(* IEC 61131-3 sources: eCockpitGit/test_project/src/%F%00 Library/%F%JSON/%POU%FB_JSONReader/%F%Read, 13 files *)

(* ---- %METH%compareString.st ---- *)
//Returns true if the inputted string is the same as the read string
METHOD compareString : BOOL
VAR_INPUT
	str				:POINTER TO EASCII;
END_VAR
VAR
	posBuffer		:POINTER TO EASCII := lastValueStart + 1;		//Buffer for key position
END_VAR
(*%!%__DELIMITER__%!%*)
IF ready AND_THEN lastValueType = EStructType.tString THEN
	WHILE posBuffer <= bufferADRMax DO
		CASE posBuffer^ OF
			EASCII.Null:
				compareString			:=		str^ = EASCII.Null;
				EXIT;
			EASCII.DoubleQoute:
				IF checkNoBackSlash(checkPos:=posBuffer) THEN
					compareString		:=		str^ = EASCII.Null;
					EXIT;
				END_IF
		END_CASE
		IF str^ <> posBuffer^ THEN
			IF posBuffer^ = EASCII.BackSlash THEN
				posBuffer				:=		posBuffer + 1;
				IF str^ <> posBuffer^ THEN
					EXIT;
				END_IF
			ELSE
				EXIT;
			END_IF
		END_IF
		str								:=		str + 1;
		posBuffer						:=		posBuffer + 1;
	END_WHILE
END_IF

(* ---- %METH%exportValue.st ---- *)
//This method outputs the start address and size of the current value
//True when ok
// |**Version**|**Author**| **Date** |**Changes**
// | 1         | NSN      | 04-06-18 | Creation
METHOD exportValue : BOOL
VAR_OUTPUT
	position		:POINTER TO EASCII;
	size			:DWORD;
END_VAR
VAR
	inString		:BOOL;
	posBuffer		:POINTER TO EASCII := lastValueStart;
	level			:WORD := 1;		//This value makes sure it doesn't return a key from inside another object
END_VAR
(*%!%__DELIMITER__%!%*)
IF ready AND lastValueStart <> 0 THEN
	position					:=		lastValueStart;
	WHILE posBuffer < bufferADRMax DO
		CASE posBuffer^ OF
			EASCII.Null:
				EXIT;
			EASCII.DoubleQoute:
				IF checkNoBackSlash(checkPos:=posBuffer) THEN
					inString	:=		NOT(inString);
				END_IF
			EASCII.CloseBraces,EASCII.SqBracketC:
				IF NOT(inString) THEN
					IF level > 1 THEN
						level	:=		level - 1;
					ELSE
						EXIT;
					END_IF
				END_IF
			EASCII.Comma:
				IF NOT(inString) THEN
					IF level <= 1 THEN
						EXIT;
					END_IF
				END_IF
			EASCII.OpenBraces,EASCII.SqBracketO:
				IF NOT(inString) THEN
					level		:=		level + 1;
				END_IF
		END_CASE
		posBuffer				:=		posBuffer + 1;
	END_WHILE
	size						:=		posBuffer - position;
	exportValue					:=		TRUE;
END_IF

(* ---- %METH%readBool.st ---- *)
METHOD readBool :BOOL
VAR
	valueBuff	:STRING(30);
END_VAR
(*%!%__DELIMITER__%!%*)
IF ready THEN
	CASE lastValueType OF
		EStructType.tBool:
			readBool				:=		lastValueStart^ = EASCII.Smallt;
		EStructType.number:
			readString(str:=ADR(valueBuff),lenMax:=30);
			readBool				:=		TO_BOOL(TO_REAL(valueBuff));
		EStructType.null:;
		EStructType.object,EStructType.tArray:
			readBool				:=		amountInSelection > 0;
		EStructType.tString:
			readString(str:=ADR(valueBuff),lenMax:=5);
			readBool				:=		TO_BOOL(valueBuff);
			IF NOT(readBool) THEN
				readBool			:=		valueBuff[0] <> 0;
			END_IF
	END_CASE
END_IF

(* ---- %METH%readByte.st ---- *)
METHOD readByte : BYTE
VAR
	buffer		:STRING(30);
	posBuffer	:POINTER TO EASCII := lastValueStart;		//Buffer for key position
	i			:BYTE;
END_VAR
(*%!%__DELIMITER__%!%*)
IF ready THEN
	CASE lastValueType OF
		EStructType.tBool:
			IF lastValueStart^ = EASCII.Smallt THEN
				readByte			:=		1;
			END_IF
		EStructType.number:
			WHILE posBuffer <= bufferADRMax AND i < 31 DO
				CASE posBuffer^ OF
					EASCII.Zero,EASCII.One,EASCII.Two,EASCII.Three,EASCII.Four,EASCII.Five,EASCII.Six,EASCII.Seven,EASCII.Eight,EASCII.Nine:;
				ELSE
					EXIT;
				END_CASE
				buffer[i]			:=		posBuffer^;
				posBuffer			:=		posBuffer + 1;
				i					:=		i + 1;
			END_WHILE
			buffer[i]				:=		EASCII.Null;
			readByte				:=		TO_BYTE(buffer);
		EStructType.null,EStructType.object,EStructType.tArray:;
		EStructType.tString:
			readString(str:=ADR(buffer),lenMax:=30);
			readByte				:=		TO_BYTE(buffer);
	END_CASE
END_IF

(* ---- %METH%readDint.st ---- *)
METHOD readDint : DINT
VAR
	buffer		:STRING(30);
	posBuffer	:POINTER TO EASCII := lastValueStart;		//Buffer for key position
	i			:BYTE;
END_VAR
(*%!%__DELIMITER__%!%*)
IF ready THEN
	CASE lastValueType OF
		EStructType.tBool:
			IF lastValueStart^ = EASCII.Smallt THEN
				readDint			:=		1;
			END_IF
		EStructType.number:
			WHILE posBuffer <= bufferADRMax AND i < 31 DO
				CASE posBuffer^ OF
					EASCII.Zero,EASCII.One,EASCII.Two,EASCII.Three,EASCII.Four,EASCII.Five,EASCII.Six,EASCII.Seven,EASCII.Eight,EASCII.Nine,EASCII.Minus:;
				ELSE
					EXIT;
				END_CASE
				buffer[i]			:=		posBuffer^;
				posBuffer			:=		posBuffer + 1;
				i					:=		i + 1;
			END_WHILE
			buffer[i]				:=		EASCII.Null;
			readDint				:=		TO_DINT(buffer);
		EStructType.null,EStructType.object,EStructType.tArray:;
		EStructType.tString:
			readString(str:=ADR(buffer),lenMax:=30);
			readDint				:=		TO_DINT(buffer);
	END_CASE
END_IF

(* ---- %METH%readDword.st ---- *)
METHOD readDword : DWORD
VAR
	buffer		:STRING(30);
	posBuffer	:POINTER TO EASCII := lastValueStart;		//Buffer for key position
	i			:BYTE;
END_VAR
(*%!%__DELIMITER__%!%*)
IF ready THEN
	CASE lastValueType OF
		EStructType.tBool:
			IF lastValueStart^ = EASCII.Smallt THEN
				readDword			:=		1;
			END_IF
		EStructType.number:
			WHILE posBuffer <= bufferADRMax AND i < 31 DO
				CASE posBuffer^ OF
					EASCII.Zero,EASCII.One,EASCII.Two,EASCII.Three,EASCII.Four,EASCII.Five,EASCII.Six,EASCII.Seven,EASCII.Eight,EASCII.Nine:;
				ELSE
					EXIT;
				END_CASE
				buffer[i]			:=		posBuffer^;
				posBuffer			:=		posBuffer + 1;
				i					:=		i + 1;
			END_WHILE
			buffer[i]				:=		EASCII.Null;
			readDword				:=		TO_DWORD(buffer);
		EStructType.null,EStructType.object,EStructType.tArray:;
		EStructType.tString:
			readString(str:=ADR(buffer),lenMax:=30);
			readDword				:=		TO_DWORD(buffer);
	END_CASE
END_IF

(* ---- %METH%readInt.st ---- *)
METHOD readInt : INT
VAR
	buffer		:STRING(30);
	posBuffer	:POINTER TO EASCII := lastValueStart;		//Buffer for key position
	i			:BYTE;
END_VAR
(*%!%__DELIMITER__%!%*)
IF ready THEN
	CASE lastValueType OF
		EStructType.tBool:
			IF lastValueStart^ = EASCII.Smallt THEN
				readInt				:=		1;
			END_IF
		EStructType.number:
			WHILE posBuffer <= bufferADRMax AND i < 31 DO
				CASE posBuffer^ OF
					EASCII.Zero,EASCII.One,EASCII.Two,EASCII.Three,EASCII.Four,EASCII.Five,EASCII.Six,EASCII.Seven,EASCII.Eight,EASCII.Nine,EASCII.Minus:;
				ELSE
					EXIT;
				END_CASE
				buffer[i]			:=		posBuffer^;
				posBuffer			:=		posBuffer + 1;
				i					:=		i + 1;
			END_WHILE
			buffer[i]				:=		EASCII.Null;
			readInt					:=		TO_INT(buffer);
		EStructType.null,EStructType.object,EStructType.tArray:;
		EStructType.tString:
			readString(str:=ADR(buffer),lenMax:=30);
			readInt					:=		TO_INT(buffer);
	END_CASE
END_IF

(* ---- %METH%readLint.st ---- *)
METHOD readLint : LINT
VAR
	buffer		:STRING(30);
	posBuffer	:POINTER TO EASCII := lastValueStart;		//Buffer for key position
	i			:BYTE;
END_VAR
(*%!%__DELIMITER__%!%*)
IF ready THEN
	CASE lastValueType OF
		EStructType.tBool:
			IF lastValueStart^ = EASCII.Smallt THEN
				readLint			:=		1;
			END_IF
		EStructType.number:
			WHILE posBuffer <= bufferADRMax AND i < 31 DO
				CASE posBuffer^ OF
					EASCII.Zero,EASCII.One,EASCII.Two,EASCII.Three,EASCII.Four,EASCII.Five,EASCII.Six,EASCII.Seven,EASCII.Eight,EASCII.Nine,EASCII.Minus:;
				ELSE
					EXIT;
				END_CASE
				buffer[i]			:=		posBuffer^;
				posBuffer			:=		posBuffer + 1;
				i					:=		i + 1;
			END_WHILE
			buffer[i]				:=		EASCII.Null;
			readLint				:=		TO_LINT(buffer);
		EStructType.null,EStructType.object,EStructType.tArray:;
		EStructType.tString:
			readString(str:=ADR(buffer),lenMax:=30);
			readLint				:=		TO_LINT(buffer);
	END_CASE
END_IF

(* ---- %METH%readLword.st ---- *)
METHOD readLword : LWORD
VAR
	buffer		:STRING(30);
	posBuffer	:POINTER TO EASCII := lastValueStart;		//Buffer for key position
	i			:BYTE;
END_VAR
(*%!%__DELIMITER__%!%*)
IF ready THEN
	CASE lastValueType OF
		EStructType.tBool:
			IF lastValueStart^ = EASCII.Smallt THEN
				readLword			:=		1;
			END_IF
		EStructType.number:
			WHILE posBuffer <= bufferADRMax AND i < 31 DO
				CASE posBuffer^ OF
					EASCII.Zero,EASCII.One,EASCII.Two,EASCII.Three,EASCII.Four,EASCII.Five,EASCII.Six,EASCII.Seven,EASCII.Eight,EASCII.Nine:;
				ELSE
					EXIT;
				END_CASE
				buffer[i]			:=		posBuffer^;
				posBuffer			:=		posBuffer + 1;
				i					:=		i + 1;
			END_WHILE
			buffer[i]				:=		EASCII.Null;
			readLword				:=		TO_LWORD(buffer);
		EStructType.null,EStructType.object,EStructType.tArray:;
		EStructType.tString:
			readString(str:=ADR(buffer),lenMax:=30);
			readLword				:=		TO_LWORD(buffer);
	END_CASE
END_IF

(* ---- %METH%readReal.st ---- *)
METHOD readReal : REAL
VAR
	buffer		:STRING(30);
	posBuffer	:POINTER TO EASCII := lastValueStart;		//Buffer for key position
	i			:BYTE;
END_VAR
(*%!%__DELIMITER__%!%*)
IF ready THEN
	CASE lastValueType OF
		EStructType.tBool:
			IF lastValueStart^ = EASCII.Smallt THEN
				readReal			:=		1;
			END_IF
		EStructType.number:
			WHILE posBuffer <= bufferADRMax AND i < 31 DO
				CASE posBuffer^ OF
					EASCII.Zero,EASCII.One,EASCII.Two,EASCII.Three,EASCII.Four,EASCII.Five,EASCII.Six,EASCII.Seven,EASCII.Eight,EASCII.Nine,EASCII.Minus,EASCII.Dot,EASCII.Smalle,EASCII.BigE,EASCII.Plus:;
				ELSE
					EXIT;
				END_CASE
				buffer[i]			:=		posBuffer^;
				posBuffer			:=		posBuffer + 1;
				i					:=		i + 1;
			END_WHILE
			buffer[i]				:=		EASCII.Null;
			readReal				:=		TO_REAL(buffer);
		EStructType.null,EStructType.object,EStructType.tArray:;
		EStructType.tString:
			readString(str:=ADR(buffer),lenMax:=30);
			readReal				:=		TO_REAL(buffer);
	END_CASE
END_IF

(* ---- %METH%readString.st ---- *)
METHOD readString
VAR_INPUT
	str				:POINTER TO EASCII;		//Address of the buffer to write the string to
	lenMax			:DWORD;					//Max lenght of the buffer
END_VAR
VAR_OUTPUT
	len				:WORD;
END_VAR
VAR
	posBuffer		:POINTER TO EASCII;		//Buffer for key position
	utfFix			:POINTER TO EASCII;
	inString		:BOOL;
	level			:WORD := 1;		//This value makes sure it doesn't return a key from inside another object
END_VAR
(*%!%__DELIMITER__%!%*)
IF ready AND_THEN lastValueType <> EStructType.none THEN
	CASE lastValueType OF
		EStructType.tArray,EStructType.object:
			posBuffer				:=		lastValueStart;
			WHILE posBuffer <= bufferADRMax AND lenMax > 0 DO
				CASE posBuffer^ OF
					EASCII.Null:
						EXIT;
					EASCII.DoubleQoute:
						IF checkNoBackSlash(checkPos:=posBuffer) THEN
							inString	:=		NOT(inString);
						END_IF
					EASCII.CloseBraces,EASCII.SqBracketC:
						IF NOT(inString) THEN
							IF level > 1 THEN
								level	:=		level - 1;
							ELSE
								EXIT;
							END_IF
						END_IF
					EASCII.Comma:
						IF NOT(inString) THEN
							IF level <= 1 THEN
								EXIT;
							END_IF
						END_IF
					EASCII.OpenBraces,EASCII.SqBracketO:
						IF NOT(inString) THEN
							level		:=		level + 1;
						END_IF
				END_CASE
				str^				:=		posBuffer^;
				str					:=		str + 1;
				posBuffer			:=		posBuffer + 1;
				lenMax				:=		lenMax - 1;
			END_WHILE
			len						:=		TO_WORD(posBuffer - lastValueStart - 1);
			str^					:=		EASCII.Null;
		EStructType.number,EStructType.tBool,EStructType.null:
			posBuffer				:=		lastValueStart;
			WHILE posBuffer <= bufferADRMax AND lenMax > 0 DO
				CASE posBuffer^ OF
					EASCII.CloseBraces,EASCII.SqBracketC,EASCII.Comma,EASCII.Null:EXIT;
				END_CASE
				str^				:=		posBuffer^;
				str					:=		str + 1;
				posBuffer			:=		posBuffer + 1;
				lenMax				:=		lenMax - 1;
			END_WHILE
			len						:=		TO_WORD(posBuffer - lastValueStart - 1);
			str^					:=		EASCII.Null;
		EStructType.tString:
			posBuffer				:=		lastValueStart + 1;
			WHILE posBuffer <= bufferADRMax AND lenMax > 0 DO
				CASE posBuffer^ OF
					EASCII.Null:EXIT;
					EASCII.DoubleQoute:
						IF checkNoBackSlash(checkPos:=posBuffer) THEN
							EXIT;
						ELSE
							str		:=		str - 1;
						END_IF
				END_CASE
				str^				:=		posBuffer^;
				str					:=		str + 1;
				posBuffer			:=		posBuffer + 1;
				lenMax				:=		lenMax - 1;
			END_WHILE
			len						:=		TO_WORD(posBuffer - lastValueStart - 1);
			str^					:=		EASCII.Null;
			CASE FU_CheckUTF8(strStart:=str - len,char:=str - 1, start=>utfFix) OF
				1,2,4:
					utfFix^			:=		0;
					len				:=		len - TO_WORD(str - utfFix);
			END_CASE
	END_CASE
END_IF

(* ---- %METH%readStringLen.st ---- *)
//This method returns the lenght of the the currently selected string
//Returns true on output if length is valid
METHOD readStringLen : WORD
VAR
	posBuffer		:POINTER TO EASCII;		//Buffer for key position
	inString		:BOOL;
	level			:WORD := 1;		//This value makes sure it doesn't return a key from inside another object
END_VAR
(*%!%__DELIMITER__%!%*)
IF ready AND_THEN lastValueType <> EStructType.none THEN
	CASE lastValueType OF
		EStructType.tArray,EStructType.object:
			posBuffer					:=		lastValueStart;
			WHILE posBuffer <= bufferADRMax DO
				CASE posBuffer^ OF
					EASCII.Null:
						EXIT;
					EASCII.DoubleQoute:
						IF checkNoBackSlash(checkPos:=posBuffer) THEN
							inString	:=		NOT(inString);
						END_IF
					EASCII.CloseBraces,EASCII.SqBracketC:
						IF NOT(inString) THEN
							IF level > 1 THEN
								level	:=		level - 1;
							ELSE
								EXIT;
							END_IF
						END_IF
					EASCII.Comma:
						IF NOT(inString) THEN
							IF level <= 1 THEN
								EXIT;
							END_IF
						END_IF
					EASCII.OpenBraces,EASCII.SqBracketO:
						IF NOT(inString) THEN
							level		:=		level + 1;
						END_IF
				END_CASE
				posBuffer				:=		posBuffer + 1;
			END_WHILE
			readStringLen				:=		TO_WORD(posBuffer - lastValueStart - 1);
		EStructType.number,EStructType.tBool,EStructType.null:
			posBuffer					:=		lastValueStart;
			WHILE posBuffer <= bufferADRMax DO
				CASE posBuffer^ OF
					EASCII.CloseBraces,EASCII.SqBracketC,EASCII.Comma,EASCII.Null:EXIT;
				END_CASE
				posBuffer				:=		posBuffer + 1;
			END_WHILE
			readStringLen				:=		TO_WORD(posBuffer - lastValueStart - 1);
		EStructType.tString:
			WHILE posBuffer <= bufferADRMax DO
				CASE posBuffer^ OF
					EASCII.Null:EXIT;
					EASCII.DoubleQoute:
						IF checkNoBackSlash(checkPos:=posBuffer) THEN
							EXIT;
						END_IF
				END_CASE
				posBuffer				:=		posBuffer + 1;
			END_WHILE
			readStringLen				:=		TO_WORD(posBuffer - lastValueStart - 1);
	END_CASE
END_IF

(* ---- %METH%readWord.st ---- *)
METHOD readWord : WORD
VAR
	buffer		:STRING(30);
	posBuffer	:POINTER TO EASCII := lastValueStart;		//Buffer for key position
	i			:BYTE;
END_VAR
(*%!%__DELIMITER__%!%*)
IF ready THEN
	CASE lastValueType OF
		EStructType.tBool:
			IF lastValueStart^ = EASCII.Smallt THEN
				readWord			:=		1;
			END_IF
		EStructType.number:
			WHILE posBuffer <= bufferADRMax AND i < 31 DO
				CASE posBuffer^ OF
					EASCII.Zero,EASCII.One,EASCII.Two,EASCII.Three,EASCII.Four,EASCII.Five,EASCII.Six,EASCII.Seven,EASCII.Eight,EASCII.Nine:;
				ELSE
					EXIT;
				END_CASE
				buffer[i]			:=		posBuffer^;
				posBuffer			:=		posBuffer + 1;
				i					:=		i + 1;
			END_WHILE
			buffer[i]				:=		EASCII.Null;
			readWord				:=		TO_WORD(buffer);
		EStructType.null,EStructType.object,EStructType.tArray:;
		EStructType.tString:
			readString(str:=ADR(buffer),lenMax:=30);
			readWord				:=		TO_WORD(buffer);
	END_CASE
END_IF
